INTERFACE I_NciChannel

(*
===============================================================
Implementation of Tc2_NCI.CfgBuildExt3DGroup

  Builds complete NCI-Group with all configured axes
===============================================================
*)
METHOD BuildGroup : HRESULT
VAR_INPUT
  Execute: BOOL;
END_VAR
END_METHOD

(*
===============================================================
NCI-Group configured axes structure
===============================================================
*)
PROPERTY CfgAxes : Tc2_NCI.NCI_EXT3DGROUP
SET
END_SET
END_PROPERTY

(*
===============================================================
Implementation of Tc2_NCI.CfgReconfigGroup

  remove all axes from NCI-Group
===============================================================
*)
METHOD ClearGroup : HRESULT
VAR_INPUT
  Execute: BOOL;
END_VAR
END_METHOD

METHOD ConfirmHSK : HRESULT
VAR_INPUT
  Execute: BOOL;
END_VAR
END_METHOD

(*
===============================================================
Implementation of Tc2_NCI.ItpDelDtgEx

  DelDTG ( delete distance to go ) wird aus dem NC Programm satzweise aktiviert. 
  Dieses Kommando ermöglicht es, aus der SPS ( TcNci.lib ItpDelDtgEx) den Restweg der aktuellen Geometrie zu löschen. 
  D.h. trifft das Kommando während der Abarbeitung des Satzes ein so wird mit den üblichen Verzögerungsrampen die Bewegung angehalten. 
  Anschließend wird mit dem nächsten Satz im NC Programm fortgefahren.
  Falls das SPS-Kommando nicht während der Ausführung eines Satzes mit angewähltem Restweglöschen eintrifft, wird dieses mit einer Fehlermeldung beantwortet.
  Das Restweglöschen bewirkt immer einen impliziten Dekodierstop, d.h. es erfolgt am Satzende immer ein Genauhalt.
===============================================================
*)
METHOD DelDTG : HRESULT
VAR_INPUT
  Execute: BOOL;
END_VAR
END_METHOD

PROPERTY Error : BOOL
GET
END_GET
END_PROPERTY

METHOD Error_Get : BOOL
END_METHOD

(*
===============================================================
Implementation of Tc2_NCI.ItpEStopEx
===============================================================
*)
METHOD EStop : HRESULT
VAR_INPUT
  Execute: BOOL;
END_VAR
END_METHOD

METHOD GetChannelOverride : real
VAR_INPUT
END_VAR
END_METHOD

METHOD GetItpState : uint
VAR_INPUT
END_VAR
END_METHOD

PROPERTY HSK : BOOL
GET
END_GET
END_PROPERTY

PROPERTY I_AuxAxis : ARRAY[1..GVL_NCI.cAuxAxisCount] OF I_McAxis
SET
END_SET
END_PROPERTY

PROPERTY I_McAxis : array[1..GVL_NCI.cMcAxisCount] of I_McAxis
SET
END_SET
END_PROPERTY

PROPERTY ItpAxes : Tc2_NCI.NCI_EXT3DGROUP
GET
END_GET
END_PROPERTY

(*
===============================================================
Implementation of Tc2_NCI.ItpResetEx2
===============================================================
*)
METHOD ItpReset : HRESULT
VAR_INPUT
  Execute: BOOL;
END_VAR
END_METHOD

METHOD LoadProg : HRESULT
VAR_INPUT
  Execute: BOOL;
END_VAR
END_METHOD

PROPERTY MFunc : INT
GET
END_GET
END_PROPERTY

PROPERTY Override : LREAL
GET
END_GET
SET
END_SET
END_PROPERTY

PROPERTY PathVelo : LREAL
GET
END_GET
END_PROPERTY

PROPERTY pNciChannelRef : POINTER TO ST_NciChannel_Ref
GET
END_GET
END_PROPERTY

PROPERTY Prog : STRING(255)
GET
END_GET
SET
END_SET
END_PROPERTY

(*
===============================================================
Implementation of Tc2_System.ADSREADEX

  reads actual interpreter G-Code Line
===============================================================
*)
METHOD ReadLine : HRESULT
VAR_INPUT
  Execute: BOOL;
END_VAR
//Read G-Code actual Line
VAR_OUTPUT
  ActProgLine: STRING(100);
END_VAR
END_METHOD

(*
===============================================================
Implementation of Tc2_NCI.ItpReadRParamsEx

  read R-Parameter(s) from NCI
===============================================================
*)
METHOD ReadRParams : HRESULT
VAR_INPUT
  Execute :BOOL;
  Addr    :POINTER TO LREAL;  //Adresse der Zielvariablen der zu lesenden Daten. 
        //Dabei werden die Daten direkt ab der angegebenen Adresse von der NC beschrieben  
        //D.h. nIndex ist nicht als Offset zu pAddr zu sehen. Die Daten befinden sich z.B. 
        //in einem Array vom Typ LREAL, das vom Anwender definiert werden muss.
  Index   :DINT;
  Count   :DINT;
END_VAR
END_METHOD

(*
===============================================================
Implementation of Tc2_NCI.ItpStartStopEx

  Start Interpreter
===============================================================
*)
METHOD StartStop : HRESULT
VAR_INPUT
  Start: BOOL;
  Stop: BOOL;
END_VAR
END_METHOD

(*
===============================================================
Implementation of Tc2_NCI.ItpStopOnAfterEStopEx
===============================================================
*)
METHOD StepOnAfterEStop : HRESULT
VAR_INPUT
  Execute: BOOL;
END_VAR
END_METHOD

(*
===============================================================
Implementation of Tc2_NCI.ItpWriteRParamsEx

  write R-Parameter(s) to NCI
===============================================================
*)
METHOD WriteRParams : HRESULT
VAR_INPUT
  Execute :BOOL;
  Addr    :POINTER TO LREAL;  //Adresse der Zielvariablen der Daten. 
        //Dabei werden die Daten direkt ab der angegebenen Adresse von der NC beschrieben  
        //D.h. nIndex ist nicht als Offset zu pAddr zu sehen. Die Daten befinden sich z.B. 
        //in einem Array vom Typ LREAL, das vom Anwender definiert werden muss.
  Index   :DINT;
  Count   :DINT;
END_VAR
END_METHOD

END_INTERFACE

(* stored: Version 1.1.0.1, ProductVersion 3.1.4024.9
   Itf I_NciChannel: Id {22099960-a888-007d-2e1b-796d477cf2b7}
   Folder methods: Id {c3bca060-2de5-0c49-3cc5-af776e588ec7}
   Folder properties: Id {809c42a6-6b4b-0217-1328-e9127f97ec50}
   Method BuildGroup: Id {a50a1117-1d46-049c-3a91-c5f7324eea07}
   Property CfgAxes: Id {03bac3e5-bb2e-00f8-235f-e0a6b4d2cc42}
   Set Set: Id {f6dc3172-31e9-093e-1a97-cc71d972586a}
   Method ClearGroup: Id {3ed05578-f813-04af-3a09-668c3202a67a}
   Method ConfirmHSK: Id {6c6d845e-e90e-05fc-2fbc-607de6a597de}
   Method DelDTG: Id {e813f933-15d9-05c8-343d-e6505f66d185}
   Property Error: Id {9ba3301d-2f33-04c1-3826-1a99022588ed}
   Get Get: Id {40612e47-1d1b-0fe6-368d-af1013a49814}
   Method Error_Get: Id {1ebeb184-4381-0df2-309b-98fe14740ac6}
   Method EStop: Id {7a3a79af-239c-0e77-1462-49de057ad951}
   Method GetChannelOverride: Id {507c7828-d40a-08fb-3ffc-744d753ed99f}
   Method GetItpState: Id {e73f2805-4dd5-46b7-86b5-e93b6c652fa8}
   Property HSK: Id {fffe650c-85ea-0c5c-15a4-0e71c3105ed4}
   Get Get: Id {621c3cb2-cfa4-0edc-2d22-92e267a999c7}
   Property I_AuxAxis: Id {22a64fdf-068b-0f49-084f-6e50e1374061}
   Set Set: Id {15a9c7f2-ccd7-0b82-38e8-98dbab1880d1}
   Property I_McAxis: Id {6c5eca0d-db81-07ea-308f-4b3fb5291003}
   Set Set: Id {cabc711a-8284-07ae-1717-283bbff8eb45}
   Property ItpAxes: Id {044da016-c642-032a-2d0d-98d36110b588}
   Get Get: Id {c74b9452-c5d8-097b-26ec-23da88bf3bea}
   Method ItpReset: Id {60785cfd-0de1-0d19-1184-86cf7ea52f52}
   Method LoadProg: Id {14bd4f28-0214-0fa4-0baa-96bb6c08927a}
   Property MFunc: Id {94450021-eb97-0b3d-2be9-62c1a02064e8}
   Get Get: Id {938436e6-e963-081a-2486-fdfab8550a3d}
   Property Override: Id {41653181-d06a-0244-0c9b-20d02894b91a}
   Get Get: Id {433480b8-b0f3-0d9a-3937-8f568c8fcbe2}
   Set Set: Id {e646ddfd-33d6-0639-3f01-fa59ed0085e5}
   Property PathVelo: Id {9ed50378-0ca4-061a-35ca-e4277fa4db5d}
   Get Get: Id {408291f9-b854-0b2e-2c20-8f8e7846f77f}
   Property pNciChannelRef: Id {85577e6e-10bf-04a6-1adc-2a2047556043}
   Get Get: Id {1351733f-88b6-081a-0e43-28544ff1d680}
   Property Prog: Id {f460be4b-8f39-0bb6-15d8-648063203c43}
   Get Get: Id {2689a867-e387-0565-0fac-30471b5aaa2e}
   Set Set: Id {47f7bf74-3095-018b-27a2-ac850438bcd0}
   Method ReadLine: Id {420751c9-bde4-06ed-13f5-c5032b61bc4f}
   Method ReadRParams: Id {3ea78807-1a7f-01a7-0d09-e9537fa77aa8}
   Method StartStop: Id {01a4af99-cc85-0f5d-12f5-596772f300cf}
   Method StepOnAfterEStop: Id {e06b7dbe-c272-0f4d-158e-66e379a8daa2}
   Method WriteRParams: Id {cf0007c8-582d-052a-106e-4fc35db440dd} *)
